(* IEC 61131-3 sources: com.logicals.lc3.webinar/usRTS_RPMControl_iSOC/src_FB_LIB_SAFE/Bitstring/DWORD, 10 files *)

(* ---- wAND_DWORD_2.iecst ---- *)
NAMESPACE logicals.web.standard
NAMESPACE bitstring

/*
 * Function block wrapper for IEC 61131-3 AND<br>
 * IN1 =  1st value (DWORD)<br>
 * IN2 =  2nd value (DWORD)<br>
 * OUT = IN1 AND IN2 (DWORD)<br>
 */
FUNCTION_BLOCK wAND_DWORD_2
	{ vNameAlignment:="center"; altName:="&"; bgColor:="DodgerBlue"; width:=40; hideIONames; }
	VAR_INPUT
		IN1 : DWORD;
		IN2 : DWORD;
	END_VAR
	VAR_OUTPUT
		OUT: DWORD;
	END_VAR

	OUT := AND(IN1:=IN1, IN2:=IN2, ENO=>ENO);
END_FUNCTION_BLOCK

END_NAMESPACE
END_NAMESPACE

(* ---- wAND_DWORD_3.iecst ---- *)
NAMESPACE logicals.web.standard
NAMESPACE bitstring

/*
 * Function block wrapper for IEC 61131-3 AND<br>
 * IN1 =  1st value (DWORD)<br>
 * IN2 =  2nd value (DWORD)<br>
 * IN3 =  3rd value (DWORD)<br>
 * OUT = IN1 AND IN2 AND IN3 (DWORD)<br>
 */
FUNCTION_BLOCK wAND_DWORD_3
	{ vNameAlignment:="center"; altName:="&"; bgColor:="DodgerBlue"; width:=40; hideIONames; }
	VAR_INPUT
		IN1 : DWORD;
		IN2 : DWORD;
		IN3 : DWORD;
	END_VAR
	VAR_OUTPUT
		OUT: DWORD;
	END_VAR

	OUT := AND(IN1:=IN1, IN2:=IN2, IN3:=IN3, ENO=>ENO);
END_FUNCTION_BLOCK

END_NAMESPACE
END_NAMESPACE

(* ---- wAND_DWORD_4.iecst ---- *)
NAMESPACE logicals.web.standard
NAMESPACE bitstring

/*
 * Function block wrapper for IEC 61131-3 AND<br>
 * IN1 =  1st value (DWORD)<br>
 * IN2 =  2nd value (DWORD)<br>
 * IN3 =  3rd value (DWORD)<br>
 * IN4 =  4th value (DWORD)<br>
 * OUT = IN1 AND IN2 AND IN3 AND IN4 (DWORD)<br>
 */
FUNCTION_BLOCK wAND_DWORD_4
	{ vNameAlignment:="center"; altName:="&"; bgColor:="DodgerBlue"; width:=40; hideIONames; }
	VAR_INPUT
		IN1 : DWORD;
		IN2 : DWORD;
		IN3 : DWORD;
		IN4 : DWORD;
	END_VAR
	VAR_OUTPUT
		OUT: DWORD;
	END_VAR

	OUT := AND(IN1:=IN1, IN2:=IN2, IN3:=IN3, IN4:=IN4, ENO=>ENO);
END_FUNCTION_BLOCK

END_NAMESPACE
END_NAMESPACE

(* ---- wNOT_DWORD.iecst ---- *)
NAMESPACE logicals.web.standard
NAMESPACE bitstring

/*
 * Function block wrapper for IEC 61131-3 NOT<br>
 * IN = input (DWORD)<br>
 * OUT = !IN (DWORD)<br>
 */
FUNCTION_BLOCK wNOT_DWORD
	{ vNameAlignment:="center"; altName:="NOT"; bgColor:="DodgerBlue"; width:=60; hideIONames; }
	VAR_INPUT
		IN : DWORD;
	END_VAR
	VAR_OUTPUT
		OUT: DWORD;
	END_VAR

	OUT := NOT(IN:=IN, ENO=>ENO);
END_FUNCTION_BLOCK

END_NAMESPACE
END_NAMESPACE

(* ---- wOR_DWORD_2.iecst ---- *)
NAMESPACE logicals.web.standard
NAMESPACE bitstring

/*
 * Function block wrapper for IEC 61131-3 OR<br>
 * IN1 =  1st value (DWORD)<br>
 * IN2 =  2nd value (DWORD)<br>
 * OUT = IN1 OR IN2 (DWORD)<br>
 */
FUNCTION_BLOCK wOR_DWORD_2
	{ vNameAlignment:="center"; altName:=">=1"; bgColor:="DodgerBlue"; width:=40; hideIONames; }
	VAR_INPUT
		IN1 : DWORD;
		IN2 : DWORD;
	END_VAR
	VAR_OUTPUT
		OUT: DWORD;
	END_VAR

	OUT := OR(IN1:=IN1, IN2:=IN2, ENO=>ENO);
END_FUNCTION_BLOCK

END_NAMESPACE
END_NAMESPACE

(* ---- wOR_DWORD_3.iecst ---- *)
NAMESPACE logicals.web.standard
NAMESPACE bitstring

/*
 * Function block wrapper for IEC 61131-3 OR<br>
 * IN1 =  1st value (DWORD)<br>
 * IN2 =  2nd value (DWORD)<br>
 * IN3 =  3rd value (DWORD)<br>
 * OUT = IN1 OR IN2 OR IN3 (DWORD)<br>
 */
FUNCTION_BLOCK wOR_DWORD_3
	{ vNameAlignment:="center"; altName:=">=1"; bgColor:="DodgerBlue"; width:=40; hideIONames; }
	VAR_INPUT
		IN1 : DWORD;
		IN2 : DWORD;
		IN3 : DWORD;
	END_VAR
	VAR_OUTPUT
		OUT: DWORD;
	END_VAR

	OUT := OR(IN1:=IN1, IN2:=IN2, IN3:=IN3, ENO=>ENO);
END_FUNCTION_BLOCK

END_NAMESPACE
END_NAMESPACE

(* ---- wOR_DWORD_4.iecst ---- *)
NAMESPACE logicals.web.standard
NAMESPACE bitstring

/*
 * Function block wrapper for IEC 61131-3 OR<br>
 * IN1 =  1st value (DWORD)<br>
 * IN2 =  2nd value (DWORD)<br>
 * IN3 =  3rd value (DWORD)<br>
 * IN4 =  4th value (DWORD)<br>
 * OUT = IN1 OR IN2 OR IN3 OR IN4 (DWORD)<br>
 */
FUNCTION_BLOCK wOR_DWORD_4
	{ vNameAlignment:="center"; altName:=">=1"; bgColor:="DodgerBlue"; width:=40; hideIONames; }
	VAR_INPUT
		IN1 : DWORD;
		IN2 : DWORD;
		IN3 : DWORD;
		IN4 : DWORD;
	END_VAR
	VAR_OUTPUT
		OUT: DWORD;
	END_VAR

	OUT := OR(IN1:=IN1, IN2:=IN2, IN3:=IN3, IN4:=IN4, ENO=>ENO);
END_FUNCTION_BLOCK

END_NAMESPACE
END_NAMESPACE

(* ---- wXOR_DWORD_2.iecst ---- *)
NAMESPACE logicals.web.standard
NAMESPACE bitstring

/*
 * Function block wrapper for IEC 61131-3 XOR<br>
 * IN1 =  1st value (DWORD)<br>
 * IN2 =  2nd value (DWORD)<br>
 * OUT = IN1 XOR IN2 (DWORD)<br>
 */
FUNCTION_BLOCK wXOR_DWORD_2
	{ vNameAlignment:="center"; altName:="=2k+1"; bgColor:="DodgerBlue"; width:=50; hideIONames; }
	VAR_INPUT
		IN1 : DWORD;
		IN2 : DWORD;
	END_VAR
	VAR_OUTPUT
		OUT: DWORD;
	END_VAR

	OUT := XOR(IN1:=IN1, IN2:=IN2, ENO=>ENO);
END_FUNCTION_BLOCK

END_NAMESPACE
END_NAMESPACE

(* ---- wXOR_DWORD_3.iecst ---- *)
NAMESPACE logicals.web.standard
NAMESPACE bitstring

/*
 * Function block wrapper for IEC 61131-3 XOR<br>
 * IN1 =  1st value (DWORD)<br>
 * IN2 =  2nd value (DWORD)<br>
 * IN3 =  3rd value (DWORD)<br>
 * OUT = IN1 XOR IN2 XOR IN3 (DWORD)<br>
 */
FUNCTION_BLOCK wXOR_DWORD_3
	{ vNameAlignment:="center"; altName:="=2k+1"; bgColor:="DodgerBlue"; width:=50; hideIONames; }
	VAR_INPUT
		IN1 : DWORD;
		IN2 : DWORD;
		IN3 : DWORD;
	END_VAR
	VAR_OUTPUT
		OUT: DWORD;
	END_VAR

	OUT := XOR(IN1:=IN1, IN2:=IN2, IN3:=IN3, ENO=>ENO);
END_FUNCTION_BLOCK

END_NAMESPACE
END_NAMESPACE

(* ---- wXOR_DWORD_4.iecst ---- *)
NAMESPACE logicals.web.standard
NAMESPACE bitstring

/*
 * Function block wrapper for IEC 61131-3 XOR<br>
 * IN1 =  1st value (DWORD)<br>
 * IN2 =  2nd value (DWORD)<br>
 * IN3 =  3rd value (DWORD)<br>
 * IN4 =  4th value (DWORD)<br>
 * OUT = IN1 XOR IN2 XOR IN3 XOR IN4 (DWORD)<br>
 */
FUNCTION_BLOCK wXOR_DWORD_4
	{ vNameAlignment:="center"; altName:="=2k+1"; bgColor:="DodgerBlue"; width:=50; hideIONames; }
	VAR_INPUT
		IN1 : DWORD;
		IN2 : DWORD;
		IN3 : DWORD;
		IN4 : DWORD;
	END_VAR
	VAR_OUTPUT
		OUT: DWORD;
	END_VAR

	OUT := XOR(IN1:=IN1, IN2:=IN2, IN3:=IN3, IN4:=IN4, ENO=>ENO);
END_FUNCTION_BLOCK

END_NAMESPACE
END_NAMESPACE
